Staubli VAL3: getDistance.pgx

public program getDistance(tool x_tTool, num& x_nDistance[], bool x_bCycle, num x_nIndex)
  local num l_nDistance
  local point l_pPoint
  local num l_nValue
  local trsf l_trsfEmpty
  local point l_pActual
  local point l_pPrev
begin
  // first point
  if x_bCycle
    // an other one
    //
    // get the point
    //
    l_pActual=pt:tTraj[sTrajCycle].tData[x_nIndex].pPoint
    // point
    x_nDistance=distance(l_pActual.trsf,pt:tTraj[sTrajCycle].trAppro[1])
  else
    l_pActual=pEditPoint.tData[x_nIndex].pPoint
    // point
    x_nDistance=distance(l_pActual.trsf,pt:tTraj[sTrajCycle].trDepart[1])
  endIf
end
